(* Called to attempt to keep the laser on as long as safely possible in the event of an Ion Pump failure *)
FUNCTION_BLOCK FB_SwitchboxIonPumpFailure EXTENDS FB_MaintainLaserOperation
VAR_INPUT
END_VAR
VAR_OUTPUT
END_VAR
VAR
	fbVentSwitchbox: FB_VentSwitchbox;
END_VAR

SUPER^(iq_sMessageBuffer := iq_sMessageBuffer);

CASE eStep OF
E_OpStep.IDLE: // Do nothing

E_OpStep.START: // Turn on roughing pump
	M_RunTimeoutTimer(PUMP_TIMEOUT);
	M_SetMessage('Turning on roughing pump');
	
	GVL_BTS_VAC.fb_PP_PTM.M_Run(TRUE);
	
	IF GVL_BTS_VAC.fb_PP_PTM.iq_stPTM.eState = E_PumpState.pumpRUNNING THEN
		M_ResetTimeoutTimer();
		M_SetMessage('Turning off pumping station ion pump');
		eStep := E_OpStep.BOIP_TURN_OFF_ION_PUMP;
	END_IF
	
E_OpStep.BOIP_TURN_OFF_ION_PUMP:
	M_RunTimeoutTimer(PUMP_TIMEOUT);
	GVL_BTS_VAC.fb_PP_PIP.M_Run(FALSE);
	
	IF NOT GVL_BTS_VAC.fb_PP_PIP.i_xSP_DI THEN
		M_ResetTimeoutTimer();
		IF ABS(GVL_BTS_VAC.fb_PP_GPI_1.PG.rPRESS - GVL_BTS_VAC.fb_DP_GPI.PG.rPRESS) < 1E-4 THEN
			M_SetMessage('Opening pump station valve');
			eStep := E_OpStep.BOIP_OPEN_SB_VALVE;
		ELSE
			M_SetMessage('Unable to maintain vacuum');
			M_ShutdownLaser();
			eStep := E_OpStep.BOIP_VENT_SB;
		END_IF
	END_IF
	
E_OpStep.BOIP_OPEN_SB_VALVE:
	M_RunTimeoutTimer(VALVE_TIMEOUT);
	GVL_BTS_VAC.fb_PP_VGC.M_Set_OPN_SW(TRUE);
	
	IF GVL_BTS_VAC.fb_PP_VGC.M_IsOpen() THEN
		M_ResetTimeoutTimer();
		M_SetMessage('Maintaining vacuum');
		eStep := E_OpStep.BOIP_HOLD;
	END_IF
	
E_OpStep.BOIP_HOLD:
	// Hold vacuum as long as possible.
	IF GVL_BTS_VAC.fb_DP_GCC.IG.rPRESS > 1E-4 THEN
		// Shutdown laser
		M_ShutdownLaser();
		M_SetMessage('Vacuum lost. Closing transport tubes');
		eStep := E_OpStep.BOIP_CLOSE_TRANSPORT_TUBE_VALVES;
	END_IF

E_OpStep.BOIP_CLOSE_TRANSPORT_TUBE_VALVES:
	M_RunTimeoutTimer(VALVE_TIMEOUT);
	M_CloseAllTransportTubeValves();
	
	IF M_AllTransportTubeValvesClosed() THEN
		M_ResetTimeoutTimer();
		M_SetMessage('Closing switchbox valve');
		eStep := E_OpStep.BOIP_CLOSE_SB_VALVE;
	END_IF
	
E_OpStep.BOIP_CLOSE_SB_VALVE:
	M_RunTimeoutTimer(VALVE_TIMEOUT);
	GVL_BTS_VAC.fb_PP_VGC.M_Set_OPN_SW(FALSE);
	
	IF GVL_BTS_VAC.fb_PP_VGC.M_IsClosed() THEN
		M_ResetTimeoutTimer();
		M_SetMessage('Turning off switchbox pumps');
		eStep := E_OpStep.BOIP_TURN_OFF_PUMPS;
	END_IF

E_OpStep.BOIP_TURN_OFF_PUMPS:
	M_RunTimeoutTimer(PUMP_TIMEOUT);
	GVL_BTS_VAC.fb_PP_PTM.M_Run(FALSE);
	GVL_BTS_VAC.fb_PP_PMF.M_Run(FALSE);

	IF GVL_BTS_VAC.fb_PP_PTM.iq_stPTM.eState = E_PumpState.pumpSTOPPED AND GVL_BTS_VAC.fb_PP_PMF.q_stPump.eState = E_PumpState.pumpSTOPPED THEN
		M_ResetTimeoutTimer();
		M_SetMessage('Closing pump station valves');
		eStep := E_OpStep.BOIP_CLOSE_PP_VALVES;
	END_IF

E_OpStep.BOIP_CLOSE_PP_VALVES:
	M_RunTimeoutTimer(VALVE_TIMEOUT);
	GVL_BTS_VAC.fb_PP_VRC_1.M_Set_OPN_SW(FALSE);
	GVL_BTS_VAC.fb_PP_VRC_2.M_Set_OPN_SW(FALSE);
	
	IF GVL_BTS_VAC.fb_PP_VRC_1.iq_stValve.eState = E_ValvePositionState.CLOSED AND GVL_BTS_VAC.fb_PP_VRC_2.iq_stValve.eState = E_ValvePositionState.CLOSED THEN
		M_ResetTimeoutTimer();
		M_SetMessage('Venting switchbox');
		eStep := E_OpStep.BOIP_VENT_SB;	
	END_IF
	
E_OpStep.BOIP_VENT_SB:
	M_DeferCancel(TRUE);
	fbVentSwitchbox(i_bExecute := TRUE,
		i_bCancel := i_bCancel,
		iq_sMessageBuffer := iq_sMessageBuffer);
		
	IF fbVentSwitchbox.q_bError THEN
		M_DeferCancel(FALSE);
		M_FatalError('Error while venting switchbox');
	ELSIF NOT fbVentSwitchbox.q_bBusy THEN
		M_DeferCancel(FALSE);
		M_Finish();
	END_IF
	
ELSE
	M_FatalError('Operation is in invalid state');
END_CASE

END_FUNCTION_BLOCK

(* stored: Version 1.1.0.1, ProductVersion 3.1.4022.17
   POU FB_SwitchboxIonPumpFailure: Id {58844151-53f2-4d22-a14e-02a27d7ddcbb}, SpecialFunc None *)
